DATA_BLOCK "MotorContro_DB_14"
VAR
  TON : Array[0..5] of TON_TIME;
  Zero : Array[0..15] of Bool;
END_VAR
BEGIN
END_DATA_BLOCK
